(* IEC 61131-3 sources: platform/examples/st, 2 files *)

(* ---- 01-blink-led.st ---- *)
(* ============================================================
   Blink LED — Structured Text (osoST dialect)
   Toggles a boolean every 500 ms using the millis() hardware trap.
   The classic "Hello World" of automation.
   ============================================================ *)
TRAP millis() : DINT   TRAP #12;

VAR_GLOBAL
  led  : BOOL := FALSE;
  t0   : DINT := 0;
END_VAR

PROCEDURE main()
  IF (millis() - t0) >= 500 THEN
    led := NOT led;        (* flip the state *)
    t0  := millis();       (* remember when *)
  END_IF;
  debug(led);              (* watch it blink *)
END_PROCEDURE

(* ---- 02-tank-control.st ---- *)
(* ============================================================
   Tank control — Structured Text
   Pump ON when level drops below LOW, OFF when it rises above HIGH.
   Hysteresis avoids chattering around a single set-point.
   (level_pct / pump map to osodb tags via the project's I/O bindings.)
   ============================================================ *)
VAR_GLOBAL
  level_pct : DINT := 0;      (* process value 0..100 *)
  pump      : BOOL := FALSE;  (* output *)
  low       : DINT := 20;
  high      : DINT := 80;
END_VAR

PROCEDURE main()
  IF level_pct <= low THEN
    pump := TRUE;             (* refill *)
  ELSIF level_pct >= high THEN
    pump := FALSE;            (* full *)
  END_IF;                     (* between low..high: hold state (hysteresis) *)
  debug(level_pct);
  debug(pump);
END_PROCEDURE
